// TIA Portal V17 export
// export: Created 2024-06-16T17:47:31.1688906Z, ExportSetting WithDefaults, DisplayName Totally Integrated Automation Portal, DisplayVersion V17, DisplayName TIA Portal Openness, DisplayVersion V17, DisplayName TIA Portal Version Control Interface, DisplayVersion V17, DisplayName STEP 7 Professional, DisplayVersion V17, DisplayName STEP 7 Safety, DisplayVersion V17, DisplayName WinCC Professional, DisplayVersion V17
DATA_BLOCK "St3_Out"   // DB315
{ S7_Optimized_Access := 'TRUE' }
VERSION : 0.1
// stored: AutoNumber false, DBAccessibleFromOPCUA true, DBAccessibleFromWebserver true, IsOnlyStoredInLoadMemory false, IsRetainMemResEnabled false, IsWriteProtectedInAS false, MemoryReserve 100
   VAR
      Ouverture_TrappeEntree : Bool;   // Ouverture : Trappe d'entrée
      Fermeture_TrappeEntree : Bool;   // Fermeture : Trappe de sortie
      Ouverture_TrappeSortie : Bool;   // Ouverture : Trappe de sortie
      Fermeture_TrappeSortie : Bool;   // Fermeture : Trappe de sortie
      Ouverture_Obturateur : Bool;   // Ouverture : Obturateur
      Fermeture_Obturateur : Bool;   // Fermeture : Obturateur
      Femerture_PorteRX : Bool;   // Ouverte : Porte RX (Homme)
      Ouverture_PorteRX : Bool;   // Fermeture : Porte RX (Homme)
   END_VAR
BEGIN
END_DATA_BLOCK
